// Mitsubishi GX Works2 project: 정량출수정수기   PLC: Q02U

PROGRAM MAIN
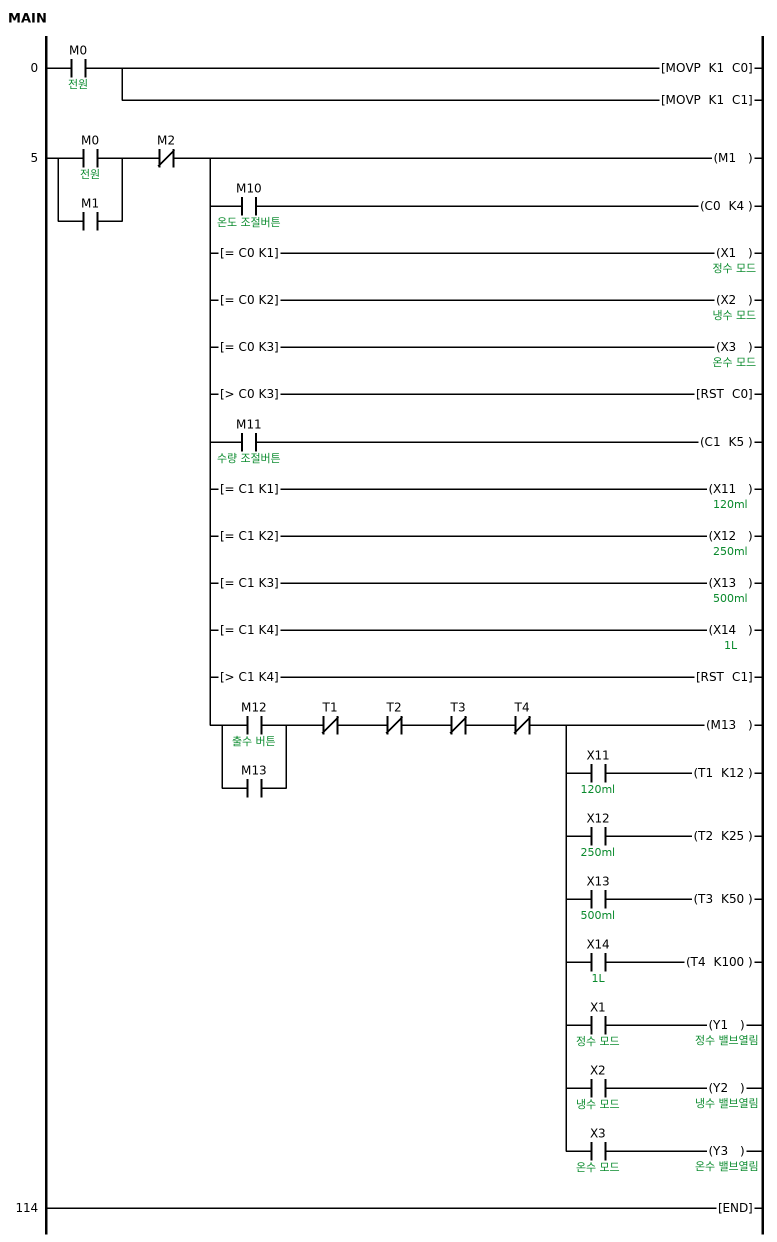
0     LD      M0  ; 전원
      MOVP    K1 C0
      MOVP    K1 C1
5     LD      M0  ; 전원
      OR      M1
      ANI     M2
      OUT     M1
      MPS
      AND     M10  ; 온도 조절버튼
      OUT     C0 K4
      MRD
      AND=    C0 K1
      OUT     X1  ; 정수 모드
      MRD
      AND=    C0 K2
      OUT     X2  ; 냉수 모드
      MRD
      AND=    C0 K3
      OUT     X3  ; 온수 모드
      MRD
      AND>    C0 K3
      RST     C0
      MRD
      AND     M11  ; 수량 조절버튼
      OUT     C1 K5
      MRD
      AND=    C1 K1
      OUT     X11  ; 120ml
      MRD
      AND=    C1 K2
      OUT     X12  ; 250ml
      MRD
      AND=    C1 K3
      OUT     X13  ; 500ml
      MRD
      AND=    C1 K4
      OUT     X14  ; 1L
      MRD
      AND>    C1 K4
      RST     C1
      MPP
      LD      M12  ; 출수 버튼
      OR      M13
      ANB
      ANI     T1
      ANI     T2
      ANI     T3
      ANI     T4
      OUT     M13
      MPS
      AND     X11  ; 120ml
      OUT     T1 K12
      MRD
      AND     X12  ; 250ml
      OUT     T2 K25
      MRD
      AND     X13  ; 500ml
      OUT     T3 K50
      MRD
      AND     X14  ; 1L
      OUT     T4 K100
      MRD
      AND     X1  ; 정수 모드
      OUT     Y1  ; 정수 밸브열림
      MRD
      AND     X2  ; 냉수 모드
      OUT     Y2  ; 냉수 밸브열림
      MPP
      AND     X3  ; 온수 모드
      OUT     Y3  ; 온수 밸브열림
114   END
END_PROGRAM
